Fanuc KAREL source: port_DOUT.kl

PROGRAM TP
%NOLOCKGROUP
VAR
 x: BOOLEAN
BEGIN
 x = DOUT[3]
END TP
